TYPE Motion_Command_Input :
STRUCT
	mode : E_6Axis_Motion;
	precise : BOOL; // 專門給Homing指令使用
	StartPOS : ARRAY [1..6] OF LREAL;
	FinalPOS : ARRAY [1..6] OF LREAL;
	
END_STRUCT
END_TYPE

(* stored: Version 1.1.0.1, ProductVersion 3.1.4024.13
   DUT Motion_Command_Input: Id {ae65b2bf-0915-4abd-917f-de52d3bce096} *)
